Staubli VAL3: Control.pgx

program Control()
begin
  //
  while true
    //急停按下：结束立即结束
    if esStatus()==2
      PublicData:sStatus="Estop"
      call StopMotion()
      bExit=true
      return
    endIf
    //endstop:单循环结束停止
    if IO:diEndStop==true
      PublicData:sStatus="endstop"
      wait(IO:diEndStop==false)
    endIf

    //start/resume
    if IO:diStart==true
      //
      if PublicData:sStatus=="stop"
        PublicData:sStatus="run"
        enablePower()
      elseIf PublicData:sStatus=="pause"
        PublicData:sStatus="run"
        restartMove()
      elseIf PublicData:sStatus=="run"
        PublicData:sStatus="pause"
        stopMove()
       endIf
      wait(IO:diStart==false)
    endIf
    delay(0)
  endWhile

end
